FUNCTION_BLOCK SampleTaskIteration EXTENDS TcoCore.TcoTask
VAR	
	_x : LREAL;
	_y : LREAL;
	_d : LREAL;
	{attribute addProperty Minimum 100}
	{attribute addProperty Maximum 1000}
	_iterations : INT;	
	_currentIteration : INT;	
END_VAR

IF(Execute()) THEN
	_y := SIN(_x);
	_x := _x + _d;		
	_currentIteration := _currentIteration + 1;	
	DoneWhen(_currentIteration >= _iterations);
END_IF

METHOD FB_init : BOOL
VAR_INPUT
	bInitRetains : BOOL; // if TRUE, the retain variables are initialized (warm start / cold start)
	bInCopyCode : BOOL;  // if TRUE, the instance afterwards gets moved into the copy code (online change)
	ParentObject : ITcoObject;
END_VAR
END_METHOD

(*~
	<docu>
		<summary>
			Restores this instance to the Ready state. Can be called explicitly or from within one of the restore mechanisms.
			<para>
				See also <see cref="PlcDocu.TcoCore.TcoTask.AutoRestorable()"/>
			</para>
		</summary>			
	</docu>	
~*)
METHOD Restore : ITcoRestorable
SUPER^.Restore();
_x := 0.0;
_y := 0.0;
_currentIteration := 0;
END_METHOD

END_FUNCTION_BLOCK

(* stored: Version 1.1.0.1, ProductVersion 3.1.4024.9
   POU SampleTaskIteration: Id {ff8ab0ff-7eb0-0983-34f1-16de82b1c941}, SpecialFunc None
   Method FB_init: Id {f3efd563-ead3-02f1-2285-17c28b9c80b4}
   Method Restore: Id {1d66f1bc-4fc9-0e1d-2089-a2db366a8b62} *)
